% RSLogix 500 project I2P Hands-On 4 - Leo Kniffen.RSS, saved by version 10.00.00.00 %
PROJECT "UNTITLED"    % processor: Bul.1763 MicroLogix 1100 Series B %

PROGRAM FILES
  LAD 2   12 rungs

DATA FILES
  O0 OUTPUT  4 elements
  I1 INPUT  6 elements
  S2 STATUS  66 elements
  B3 BINARY  1 elements
  T4 TIMER  1 elements
  C5 COUNTER  1 elements
  R6 CONTROL  1 elements
  N7 INTEGER  1 elements
  F8 FLOAT  1 elements

LADDER 2
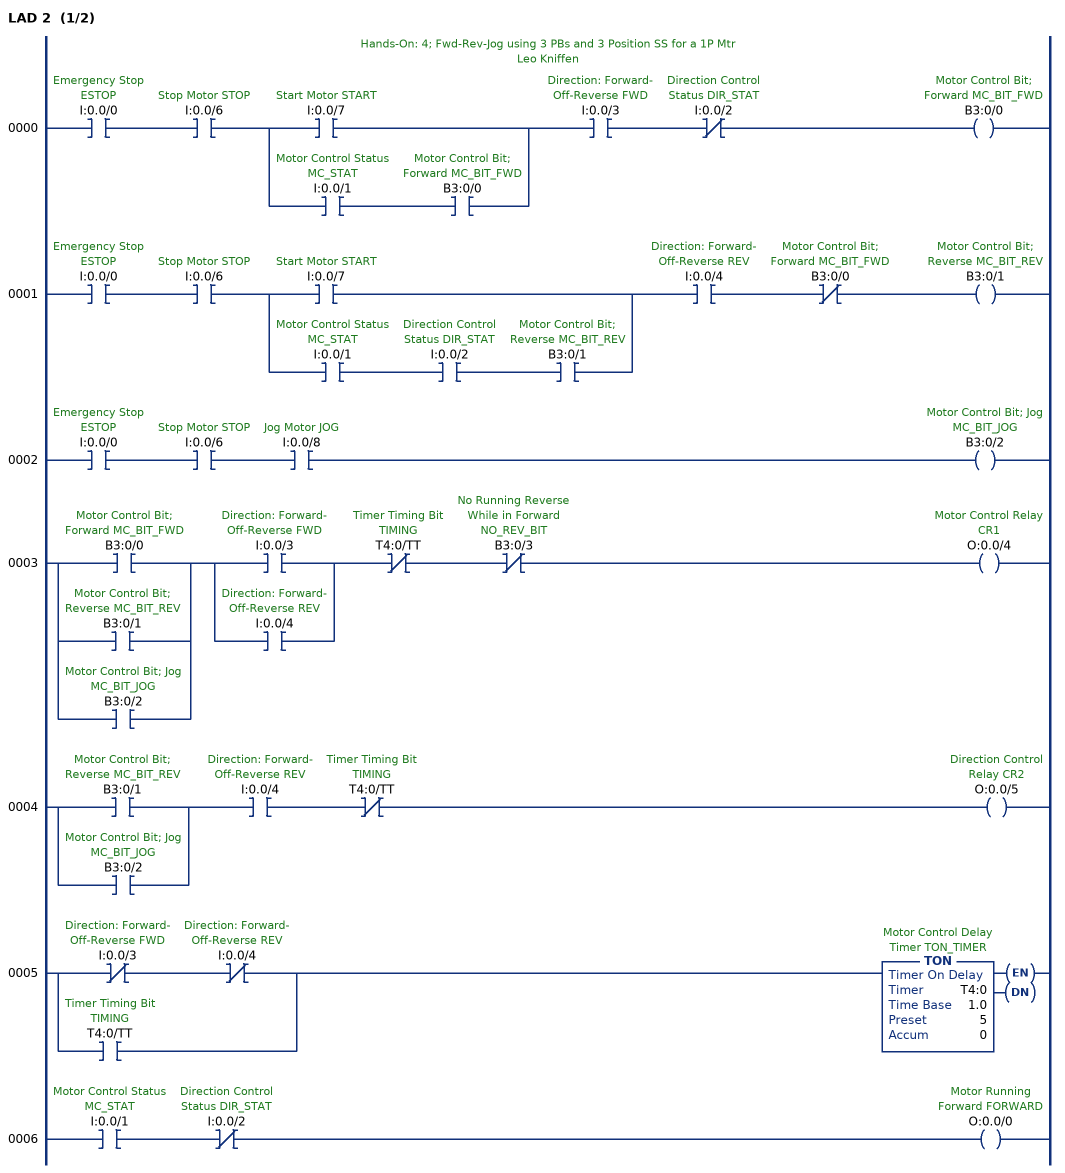
% Rung: 0 %
% Hands-On: 4; Fwd-Rev-Jog using 3 PBs and 3 Position SS for a 1P Mtr
% Leo Kniffen %
SOR XIC I:0.0/0 XIC I:0.0/6 BST XIC I:0.0/7 NXB XIC I:0.0/1 XIC B3:0/0 BND XIC I:0.0/3 XIO I:0.0/2 OTE B3:0/0 EOR
%   I:0.0/0  ESTOP  "Emergency Stop" %
%   I:0.0/6  STOP  "Stop Motor" %
%   I:0.0/7  START  "Start Motor" %
%   I:0.0/1  MC_STAT  "Motor Control Status" %
%   B3:0/0  MC_BIT_FWD  "Motor Control Bit; Forward" %
%   I:0.0/3  FWD  "Direction: Forward- Off-Reverse" %
%   I:0.0/2  DIR_STAT  "Direction Control Status" %
% Rung: 1 %
SOR XIC I:0.0/0 XIC I:0.0/6 BST XIC I:0.0/7 NXB XIC I:0.0/1 XIC I:0.0/2 XIC B3:0/1 BND XIC I:0.0/4 XIO B3:0/0 OTE B3:0/1 EOR
%   I:0.0/0  ESTOP  "Emergency Stop" %
%   I:0.0/6  STOP  "Stop Motor" %
%   I:0.0/7  START  "Start Motor" %
%   I:0.0/1  MC_STAT  "Motor Control Status" %
%   I:0.0/2  DIR_STAT  "Direction Control Status" %
%   B3:0/1  MC_BIT_REV  "Motor Control Bit; Reverse" %
%   I:0.0/4  REV  "Direction: Forward- Off-Reverse" %
%   B3:0/0  MC_BIT_FWD  "Motor Control Bit; Forward" %
% Rung: 2 %
SOR XIC I:0.0/0 XIC I:0.0/6 XIC I:0.0/8 OTE B3:0/2 EOR
%   I:0.0/0  ESTOP  "Emergency Stop" %
%   I:0.0/6  STOP  "Stop Motor" %
%   I:0.0/8  JOG  "Jog Motor" %
%   B3:0/2  MC_BIT_JOG  "Motor Control Bit; Jog" %
% Rung: 3 %
SOR BST BST XIC B3:0/0 NXB XIC B3:0/1 BND NXB XIC B3:0/2 BND BST XIC I:0.0/3 NXB XIC I:0.0/4 BND XIO T4:0/TT XIO B3:0/3 OTE O:0.0/4 EOR
%   B3:0/0  MC_BIT_FWD  "Motor Control Bit; Forward" %
%   B3:0/1  MC_BIT_REV  "Motor Control Bit; Reverse" %
%   B3:0/2  MC_BIT_JOG  "Motor Control Bit; Jog" %
%   I:0.0/3  FWD  "Direction: Forward- Off-Reverse" %
%   I:0.0/4  REV  "Direction: Forward- Off-Reverse" %
%   T4:0/TT  TIMING  "Timer Timing Bit" %
%   B3:0/3  NO_REV_BIT  "No Running Reverse While in Forward" %
%   O:0.0/4  CR1  "Motor Control Relay" %
% Rung: 4 %
SOR BST XIC B3:0/1 NXB XIC B3:0/2 BND XIC I:0.0/4 XIO T4:0/TT OTE O:0.0/5 EOR
%   B3:0/1  MC_BIT_REV  "Motor Control Bit; Reverse" %
%   B3:0/2  MC_BIT_JOG  "Motor Control Bit; Jog" %
%   I:0.0/4  REV  "Direction: Forward- Off-Reverse" %
%   T4:0/TT  TIMING  "Timer Timing Bit" %
%   O:0.0/5  CR2  "Direction Control Relay" %
% Rung: 5 %
SOR BST XIO I:0.0/3 XIO I:0.0/4 NXB XIC T4:0/TT BND TON T4:0 1.0 5 0 EOR
%   I:0.0/3  FWD  "Direction: Forward- Off-Reverse" %
%   I:0.0/4  REV  "Direction: Forward- Off-Reverse" %
%   T4:0/TT  TIMING  "Timer Timing Bit" %
%   T4:0  TON_TIMER  "Motor Control Delay Timer" %
% Rung: 6 %
SOR XIC I:0.0/1 XIO I:0.0/2 OTE O:0.0/0 EOR
%   I:0.0/1  MC_STAT  "Motor Control Status" %
%   I:0.0/2  DIR_STAT  "Direction Control Status" %
%   O:0.0/0  FORWARD  "Motor Running Forward" %

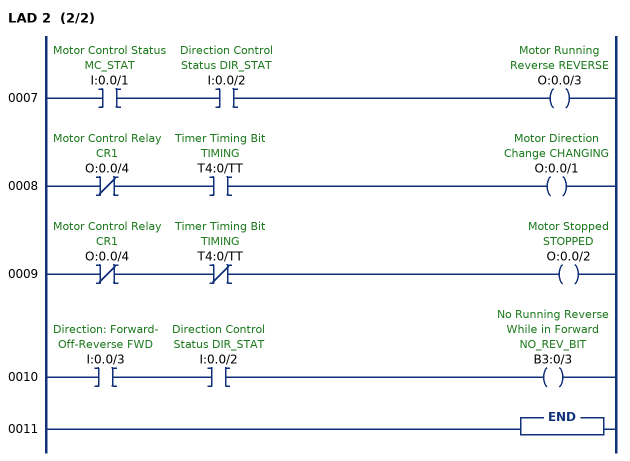
% Rung: 7 %
SOR XIC I:0.0/1 XIC I:0.0/2 OTE O:0.0/3 EOR
%   I:0.0/1  MC_STAT  "Motor Control Status" %
%   I:0.0/2  DIR_STAT  "Direction Control Status" %
%   O:0.0/3  REVERSE  "Motor Running Reverse" %
% Rung: 8 %
SOR XIO O:0.0/4 XIC T4:0/TT OTE O:0.0/1 EOR
%   O:0.0/4  CR1  "Motor Control Relay" %
%   T4:0/TT  TIMING  "Timer Timing Bit" %
%   O:0.0/1  CHANGING  "Motor Direction Change" %
% Rung: 9 %
SOR XIO O:0.0/4 XIO T4:0/TT OTE O:0.0/2 EOR
%   O:0.0/4  CR1  "Motor Control Relay" %
%   T4:0/TT  TIMING  "Timer Timing Bit" %
%   O:0.0/2  STOPPED  "Motor Stopped" %
% Rung: 10 %
SOR XIC I:0.0/3 XIC I:0.0/2 OTE B3:0/3 EOR
%   I:0.0/3  FWD  "Direction: Forward- Off-Reverse" %
%   I:0.0/2  DIR_STAT  "Direction Control Status" %
%   B3:0/3  NO_REV_BIT  "No Running Reverse While in Forward" %
% Rung: 11 %
SOR END EOR

DATA TABLE (non-zero values as saved)
DATA T4
% .PRE .ACC %
% T4:0 % 5 0
